FUNCTION_BLOCK FB_QM_Simple IMPLEMENTS IF_queueManager
VAR_INPUT
	bButtons 	  : ARRAY [1..NUMLEVELS] OF BOOL;						(* user input *)
END_VAR
VAR_OUTPUT
END_VAR
VAR
	tPushDetects  : ARRAY [1..NUMLEVELS] OF FB_BinaryInp;				(* FBs to buffer user inputs until being processed *)
	queueManip	  : FB_ArrManip;										(* FB for array manipulation, like sorting etc. *)
	k			  : INT;												(* loop variable *)
	
	nCurLevel	  : INT(1..NUMLEVELS);									(* current lift position *)
	nQueue		  : ARRAY [1..NUMLEVELS] OF INT;						(* queue, saving next targets in current moving direction *)
	bLevelInQueue : ARRAY [1..NUMLEVELS] OF BOOL;						(* buffer of all active calls , i.e. levels in nQueue OR active tPushDetects *)
END_VAR

FOR k:=1 TO NUMLEVELS DO
	tPushDetects[k](bPush:=bButtons[k], bReset:=FALSE);
	bLevelInQueue[k] := tPushDetects[k].bOutActive OR queueManip.isElement(arr:=nQueue, entry:=k);
END_FOR

FOR k:=1 TO NUMLEVELS DO
	IF tPushDetects[k].bOutActive THEN
		IF NOT queueManip.isElement(arr:=nQueue, entry:=k) THEN
			// Inset new element
			queueManip.insert(arr:=nQueue, newElement:=k, freeElement:=0);
		END_IF	
	
		// Then acknowledge
		tPushDetects[k](bReset:=TRUE);
	END_IF
END_FOR

PROPERTY currentLevel : INT (1..NUMLEVELS)
SET
nCurLevel := currentLevel;
END_SET
END_PROPERTY

METHOD doneAck
VAR_INPUT
END_VAR
VAR
END_VAR
(* 
By calling this method, the first entry in nQueue is deleted and all remaining entries are shiftetd one position forward. 
Method shall be called, after the latest moving job has been executed. 
*)
queueManip.pop_front(arr:=nQueue, fill:=0);
END_METHOD

PROPERTY queue : REFERENCE TO ARRAY [1..NUMLEVELS] OF INT
GET
queue REF= nQueue;
END_GET
END_PROPERTY

METHOD reset
VAR_INPUT
END_VAR
VAR
	i : INT;
END_VAR
(* resets all calls *)
FOR i:=1 TO NUMLEVELS DO
	nQueue[i] := 0;
	tPushDetects[i](bReset:=TRUE);
END_FOR
END_METHOD

END_FUNCTION_BLOCK

(* stored: Version 1.1.0.1, ProductVersion 3.1.4024.6
   POU FB_QM_Simple: Id {48533d12-bc5e-4f3b-a37d-0b1460f72dcd}, SpecialFunc None
   Property currentLevel: Id {05b8ddf7-4206-4f55-a2af-17307caea94c}
   Set Set: Id {4c6cbf21-05ba-409b-ab68-4544dba8e684}
   Method doneAck: Id {1917ccf5-84bb-4682-814c-910156dcf3b0}
   Property queue: Id {ff04d85a-00eb-4b9f-921f-cfd9edbf70a4}
   Get Get: Id {f1999e36-4522-4088-9557-86f50cf1d9d6}
   Method reset: Id {ba8a2664-ac75-41c1-9a13-267ab6d3bdc0} *)
